INTERFACE I_Relay

PROPERTY OFF : BOOL
GET
END_GET
END_PROPERTY

PROPERTY ON : Bool
GET
END_GET
END_PROPERTY

METHOD PUBLIC SwitchOff
VAR_INPUT
END_VAR
END_METHOD

METHOD PUBLIC SwitchOn
VAR_INPUT
END_VAR
END_METHOD

END_INTERFACE

(* stored: Version 1.1.0.1, ProductVersion 3.1.4024.15
   Itf I_Relay: Id {1984f853-e95e-423b-9025-6b27d33236a2}
   Property OFF: Id {3aca75fc-66c8-46cc-b214-83b1a558c941}
   Get Get: Id {614ecfae-0fa7-4b03-9620-7b227ea452a0}
   Property ON: Id {7650aa09-582d-4c9d-b217-946c5c288ab3}
   Get Get: Id {b340d491-20a3-4347-8461-e4635301f5ab}
   Method SwitchOff: Id {b10429bb-49f0-4f17-aaf3-788ec25870b0}
   Method SwitchOn: Id {3276d0af-d3c0-4e0a-b76c-ed8c33774338} *)
